TYPE csp_transfer_crosspusher_connection_status_enum :
(		
	CSP_TRANSFER_CROSSPUSHER_STATUS_CONNECTION_START							:= 0,
	CSP_TRANSFER_CROSSPUSHER_STATUS_CONNECTION_ENGAGE							:= 10,
	CSP_TRANSFER_CROSSPUSHER_STATUS_CONNECTION_ENGAGED							:= 20,
	CSP_TRANSFER_CROSSPUSHER_STATUS_CONNECTION_CHECK_CHANGE_CAM					:= 30,
	CSP_TRANSFER_CROSSPUSHER_STATUS_CONNECTION_CHANGE_CAM						:= 40,
	CSP_TRANSFER_CROSSPUSHER_STATUS_CONNECTION_IMMEDIATE_CHANGE					:= 45,
	CSP_TRANSFER_CROSSPUSHER_STATUS_CONNECTION_WAIT_NEW_CAM						:= 50,
	CSP_TRANSFER_CROSSPUSHER_STATUS_CONNECTION_WAIT_REJECT						:= 60,
	CSP_TRANSFER_CROSSPUSHER_STATUS_CONNECTION_WAIT_REJECT_CAM_ENGAGE			:= 65,
	CSP_TRANSFER_CROSSPUSHER_STATUS_CONNECTION_DONE 							:= 900,
	CSP_TRANSFER_CROSSPUSHER_STATUS_CONNECTION_ERROR 							:= 999
) := CSP_TRANSFER_CROSSPUSHER_STATUS_CONNECTION_START;
END_TYPE

(* stored: Version 1.1.0.1, ProductVersion 3.1.4024.3
   DUT csp_transfer_crosspusher_connection_status_enum: Id {7579c030-62c4-4739-a0a0-ded522317025} *)
